{attribute addProperty BoxType "EKM1101-0000-0016"}
{attribute addProperty Id "ControlAT %Q*Control_24A9302412115.125"}
{attribute addProperty CRC "3458699086"}
{attribute addProperty SizeInBites "121"}
{attribute addProperty SizeInBytes "15.125"}
TYPE MMS_Device_Outputs_CE278F4E :
STRUCT
	{attribute addProperty Name "Control"}
	Control AT %Q* : Control_24A93024;
END_STRUCT
END_TYPE

(* stored: Version 1.2.0.0, ProductVersion 3.1.4024.9
   DUT MMS_Device_Outputs_CE278F4E: Id {f550d9ed-b437-4ddc-92c3-10eb32db7e78} *)
